FUNCTION_BLOCK TrojanUV3000_HMI (* Service Interface Function Block Type *)
  (* Standard: 61499-2 *)
  (* Version 0.0, 03/03/2026, template *)
  PACKAGE Hidryco.HidrycoLib;
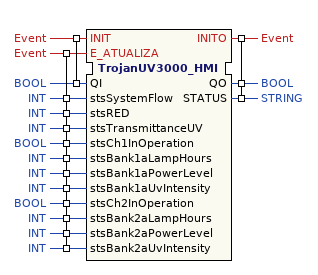
  EVENT_INPUT
    INIT WITH QI;
    E_ATUALIZA WITH stsSystemFlow, stsRED, stsTransmittanceUV, stsCh1InOperation, stsBank1aLampHours, stsBank1aPowerLevel, stsBank1aUvIntensity, stsCh2InOperation, stsBank2aLampHours, stsBank2aPowerLevel, stsBank2aUvIntensity;
  END_EVENT
  EVENT_OUTPUT
    INITO WITH QO, STATUS;
  END_EVENT
  VAR_INPUT
    QI : BOOL;
    stsSystemFlow : INT;
    stsRED : INT;
    stsTransmittanceUV : INT;
    stsCh1InOperation : BOOL;
    stsBank1aLampHours : INT;
    stsBank1aPowerLevel : INT;
    stsBank1aUvIntensity : INT;
    stsCh2InOperation : BOOL;
    stsBank2aLampHours : INT;
    stsBank2aPowerLevel : INT;
    stsBank2aUvIntensity : INT;
  END_VAR
  VAR_OUTPUT
    QO : BOOL; (* Event Output Qualifier *)
    STATUS : STRING; (* Service Status *)
  END_VAR
  SERVICE /
    SEQUENCE 
    END_SEQUENCE
  END_SERVICE
END_FUNCTION_BLOCK
